// TwinCAT 3 PLC project WorkerPLC
// ProgramVersion: 3.1.4020.4
// libraries:
//   Tc2_Standard, * (Beckhoff Automation GmbH)
//   Tc2_System, * (Beckhoff Automation GmbH)
//   Tc3_Module, * (Beckhoff Automation GmbH)
// project tree:
//   DUTs/ DigitalInput.TcDUT, DigitalOutput.TcDUT
//   / PlcTask.TcTTO
//   POUs/ MAIN.TcPOU

CONFIGURATION WorkerPLC
    RESOURCE PLC ON TwinCAT3
        TASK PlcTask(INTERVAL := T#10ms, PRIORITY := 20);
        PROGRAM MAIN WITH PlcTask : MAIN;
    END_RESOURCE
END_CONFIGURATION

// ---- DUTs/DigitalInput.TcDUT
TYPE DigitalInput :
STRUCT
	in AT %I*	:	BIT;
END_STRUCT
END_TYPE

// ---- DUTs/DigitalOutput.TcDUT
TYPE DigitalOutput :
STRUCT
	out AT %Q*	:	BIT;
END_STRUCT
END_TYPE

// ---- POUs/MAIN.TcPOU
PROGRAM MAIN
VAR
	starter	:	DigitalOutput;
	input	:	DigitalInput;
	output	:	DigitalOutput;
	term	:	DigitalInput;
END_VAR

END_PROGRAM
